      GVL_APPLICATION.Simulation[nProcess].TargetFirst   := 9;
      GVL_APPLICATION.Simulation[nProcess].TargetLast    := 9;
      GVL_APPLICATION.Simulation[nProcess].TargetMask    := 2#0001; // mask for target station

      //---------------------------------------------------------
      nProcess                                        := 9;
      tProcess[nProcess]                              := T#2200MS;

      GVL_APPLICATION.Simulation[nProcess].StationFirst  := 9;
      GVL_APPLICATION.Simulation[nProcess].StationLast   := 9;

      GVL_APPLICATION.Simulation[nProcess].TargetFirst   := 10;
      GVL_APPLICATION.Simulation[nProcess].TargetLast    := 10;
      GVL_APPLICATION.Simulation[nProcess].TargetMask    := 2#0001; // mask for target station

      //---------------------------------------------------------
      nProcess                                        := 10;
      tProcess[nProcess]                              := T#500MS;

      GVL_APPLICATION.Simulation[nProcess].StationFirst  := 10;
      GVL_APPLICATION.Simulation[nProcess].StationLast   := 10;

      GVL_APPLICATION.Simulation[nProcess].TargetFirst   := 11;
      GVL_APPLICATION.Simulation[nProcess].TargetLast    := 11;
      GVL_APPLICATION.Simulation[nProcess].TargetMask    := 2#0001; // mask for target station

      //---------------------------------------------------------
      nProcess                                        := 11;
      tProcess[nProcess]                              := T#1900MS;

      GVL_APPLICATION.Simulation[nProcess].StationFirst  := 11;
      GVL_APPLICATION.Simulation[nProcess].StationLast   := 11;

      GVL_APPLICATION.Simulation[nProcess].TargetFirst   := 12;
      GVL_APPLICATION.Simulation[nProcess].TargetLast    := 12;
      GVL_APPLICATION.Simulation[nProcess].TargetMask    := 2#0001; // mask for target station

      //---------------------------------------------------------
      nProcess                                        := 12;
      tProcess[nProcess]                              := T#2200MS;

      GVL_APPLICATION.Simulation[nProcess].StationFirst  := 12;
      GVL_APPLICATION.Simulation[nProcess].StationLast   := 12;

      GVL_APPLICATION.Simulation[nProcess].TargetFirst   := 13;
      GVL_APPLICATION.Simulation[nProcess].TargetLast    := 13;
      GVL_APPLICATION.Simulation[nProcess].TargetMask    := 2#0001; // mask for target station

      //---------------------------------------------------------
      nProcess                                        := 13;
      tProcess[nProcess]                              := T#500MS;

      GVL_APPLICATION.Simulation[nProcess].StationFirst  := 13;
      GVL_APPLICATION.Simulation[nProcess].StationLast   := 13;

      GVL_APPLICATION.Simulation[nProcess].TargetFirst   := 14;
      GVL_APPLICATION.Simulation[nProcess].TargetLast    := 15;
      GVL_APPLICATION.Simulation[nProcess].TargetMask    := 2#0001; // mask for target station

      //---------------------------------------------------------
      nProcess                                        := 14;
      tProcess[nProcess]                              := T#2000MS;

      GVL_APPLICATION.Simulation[nProcess].StationFirst  := 14;
      GVL_APPLICATION.Simulation[nProcess].StationLast   := 15;

      GVL_APPLICATION.Simulation[nProcess].TargetFirst   := 16;
      GVL_APPLICATION.Simulation[nProcess].TargetLast    := 17;
      GVL_APPLICATION.Simulation[nProcess].TargetMask    := 2#0001; // mask for target station


      //---------------------------------------------------------
      nProcess                                        := 16;
      tProcess[nProcess]                              := T#2300MS;

      GVL_APPLICATION.Simulation[nProcess].StationFirst  := 16;
      GVL_APPLICATION.Simulation[nProcess].StationLast   := 17;

      GVL_APPLICATION.Simulation[nProcess].TargetFirst   := 18;
      GVL_APPLICATION.Simulation[nProcess].TargetLast    := 18;
      GVL_APPLICATION.Simulation[nProcess].TargetMask    := 2#0001; // mask for target station

      //---------------------------------------------------------
      nProcess                                        := 18;
      tProcess[nProcess]                              := T#2200MS;

      GVL_APPLICATION.Simulation[nProcess].StationFirst  := 18;
      GVL_APPLICATION.Simulation[nProcess].StationLast   := 18;

      GVL_APPLICATION.Simulation[nProcess].TargetFirst   := 19;
      GVL_APPLICATION.Simulation[nProcess].TargetLast    := 19;
      GVL_APPLICATION.Simulation[nProcess].TargetMask    := 2#0001; // mask for target station

      //---------------------------------------------------------
      nProcess                                        := 19;
      tProcess[nProcess]                              := T#500MS;

      GVL_APPLICATION.Simulation[nProcess].StationFirst  := 19;
      GVL_APPLICATION.Simulation[nProcess].StationLast   := 19;

      GVL_APPLICATION.Simulation[nProcess].TargetFirst   := 1;
      GVL_APPLICATION.Simulation[nProcess].TargetLast    := 1;
      GVL_APPLICATION.Simulation[nProcess].TargetMask    := 2#0001; // mask for target station

    eInit                               := E_PROGRESS.PROGRESS_DONE;

END_CASE
END_ACTION

END_PROGRAM

// ---- APPLICATION/_types/LinkedList/fb_Process_LinkedListCtrl.TcPOU
FUNCTION_BLOCK fb_Process_LinkedListCtrl IMPLEMENTS I_Process_LinkedList
VAR
  _LastNodeAdded,
  _LastNodeRemoved  : ST_PROCESS_LIST_RESULT;

	_nCount           : UDINT;
  _nFree            : UDINT;

  {attribute 'hide'}
	_stList           : ARRAY[0..MAX_LIST_NODES] OF ST_PROCESS_DATA;
	_stNodes          : ARRAY[0..MAX_LIST_NODES] OF T_LinkedListEntry;

	_fbList           : Tc2_Utilities.FB_LinkedListCtrl;
	_hList            : Tc2_Utilities.T_HLINKEDLIST;

	_stRef            : POINTER TO ST_PROCESS_DATA;
END_VAR

METHOD AddHeadValue : ST_PROCESS_LIST_RESULT
VAR_INPUT
  stData        : ST_PROCESS_DATA;
END_VAR
VAR
  _nIdxNode     : ULINT; 
	_pPosGet      : POINTER TO T_LinkedListEntry;
  _stRes        : ST_PROCESS_LIST_RESULT;
END_VAR

// add empty node
_fbList.A_AddHeadValue( hList     := _hList, 
                        putValue  := 16#0, 
                        getPosPtr => _pPosGet);

IF NOT _fbList.bOk 
THEN
  _stRes.wState.0       := TRUE;
ELSE
  // Get array index of new node
	_fbList.A_GetIndexAtPosPtr( hList       := _hList, 
                              putPosPtr   := _pPosGet, 
                              getValue    => _nIdxNode);

	IF NOT _fbList.bOk 
  THEN
    _stRes.wState.1     := TRUE;
  ELSE
    // write data to new node index
		_stRef 	            := ADR( _stList[_nIdxNode] );
		_stRef^ 	          := stData;

		_fbList.A_SetValueAtPosPtr( hList     := _hList, 
                                putPosPtr := _pPosGet, 
                                putValue  := _stRef);

		IF NOT _fbList.bOk 
    THEN
      _stRes.wState.2   := TRUE;
    ELSE
      _stRes.nIndex     := _nIdxNode;
			_stRes.stData     := stData;
      _LastNodeAdded    := _stRes;
		END_IF
	END_IF
END_IF

AddHeadValue := _stRes;
END_METHOD

METHOD AddTailValue : ST_PROCESS_LIST_RESULT
VAR_INPUT
  stData        : ST_PROCESS_DATA;
END_VAR
VAR
  _nIdxNode     : ULINT; 
	_pPosGet      : POINTER TO T_LinkedListEntry;
  _stRes        : ST_PROCESS_LIST_RESULT;
END_VAR

// add empty node
_fbList.A_AddTailValue( hList       := _hList, 
                        putValue    := 16#0, 
                        getPosPtr   => _pPosGet);


IF NOT _fbList.bOk 
THEN
  _stRes.wState.0 := TRUE;
ELSE
  // Get array index of new node
	_fbList.A_GetIndexAtPosPtr( hList       := _hList, 
                              putPosPtr   := _pPosGet, 
                              getValue    => _nIdxNode);

	IF NOT _fbList.bOk 
  THEN
    _stRes.wState.1     := TRUE;
  ELSE
    // write data to new node index
		_stRef 	            := ADR( _stList[_nIdxNode] );
		_stRef^ 	          := stData;

		_fbList.A_SetValueAtPosPtr( hList     := _hList, 
                                putPosPtr := _pPosGet, 
                                putValue  := _stRef);

		IF NOT _fbList.bOk 
    THEN
      _stRes.wState.2   := TRUE;
    ELSE
      _stRes.nIndex     := _nIdxNode;
			_stRes.stData     := stData;
      _LastNodeAdded    := _stRes;
		END_IF
	END_IF
END_IF

AddTailValue := _stRes;
END_METHOD

PROPERTY Count : UDINT
GET
Count := _nCount := _hList.nCount;
END_GET
END_PROPERTY

PROPERTY Data : ARRAY[1..MAX_LIST_NODES] OF ST_PROCESS_DATA
GET
VAR
	_tList        : ARRAY[1..MAX_LIST_NODES] OF ST_PROCESS_DATA;
  _getValue     : PVOID;
  _pEntry       : POINTER TO ST_PROCESS_DATA;
  _getPosPtr    : POINTER TO T_LinkedListEntry := 0;
  _nIdx         : UINT;  
END_VAR
_fbList(
	hList       := _hList);

_nCount       := _hList.nCount;
_nFree        := _hList.nFree;


_fbList.A_GetHead( hList := _hList, getValue=> _getValue, getPosPtr=> _getPosPtr );
IF _fbList.bOk 
THEN
  IF (_hList.nCount > 0)
  THEN
    _nIdx         := 1;
    _pEntry       := _getValue;
    _tList[1]     := _pEntry^;
    
    REPEAT
      _fbList.A_GetNext( hList := _hList, putPosPtr := _getPosPtr, getValue=> _getValue, getPosPtr=> _getPosPtr );
  
      IF _fbList.bOk THEN
        _nIdx         := _nIdx + 1;
        _pEntry       := _getValue;
        _tList[_nIdx] := _pEntry^;
      ELSE
        EXIT;
      END_IF
    UNTIL NOT _fbList.bOk
    END_REPEAT
  END_IF
END_IF

Data := _tList;
END_GET
END_PROPERTY

PROPERTY Free : UDINT
GET
Free := _nFree := _hList.nFree;
END_GET
END_PROPERTY

METHOD GetHead : ST_PROCESS_LIST_RESULT
VAR_INPUT
END_VAR
VAR
	_pPosGet      : POINTER TO T_LinkedListEntry;
  _pData        : POINTER TO ST_PROCESS_DATA;
  _stRes        : ST_PROCESS_LIST_RESULT;
END_VAR

_fbList.A_GetHead(hList      := _hList,
                  getValue   => _pData,
                  getPosPtr  => _pPosGet);

IF NOT _fbList.bOk
THEN
  _stRes.wState.0 := TRUE;
ELSE
  _stRes.stData := _pData^;
END_IF

GetHead := _stRes;
END_METHOD

METHOD InitList : BOOL
VAR
  _bOk : Bool;
END_VAR

IF Tc2_Utilities.F_CreateLinkedListHnd(ADR(_stNodes), SIZEOF(_stNodes), _hList)
THEN
  _fbList.A_Reset(hList := _hList, bOk => _bOk);
  memset(ADR(_stList), 0, SIZEOF(_stList));
  _nCount   := 0;
  InitList  := TRUE; //_bOk;
END_IF
END_METHOD

PROPERTY Nodes : ARRAY[0..MAX_LIST_NODES] OF T_LinkedListEntry
GET
Nodes := _stNodes;
END_GET
END_PROPERTY

METHOD RemoveHeadValue : ST_PROCESS_LIST_RESULT
VAR_INPUT
END_VAR
VAR
	_pPosGet      : POINTER TO T_LinkedListEntry;
  _pData        : POINTER TO ST_PROCESS_DATA;
  _stRes        : ST_PROCESS_LIST_RESULT;
END_VAR
_fbList.A_RemoveHeadValue(hList       := _hList, 
                          getValue    => _pData, 
                          getPosPtr   => _pPosGet);

IF NOT _fbList.bOk 
THEN
  _stRes.wState.0 := TRUE;
ELSE
	_stRes.stData     := _pData^;
  _LastNodeRemoved  := _stRes;
  memset(_pData, 0, SIZEOF(ST_PROCESS_DATA));
END_IF
RemoveHeadValue := _stRes;
END_METHOD

END_FUNCTION_BLOCK
